FUNCTION_BLOCK FB_AllocateAreaWithRoundbelt EXTENDS FB_ModeBase_V2 IMPLEMENTS I_UnitState
VAR_INPUT
    INPUT       : REFERENCE TO ST_InputTable;
    OUTPUT      : REFERENCE TO ST_OutputTable;
    CurrentData : ST_SetupPara;
    // Componets
    Cylinder 	: REFERENCE TO UNI_CylinderList;
    Service  	: REFERENCE TO ST_AllocateService;
    Motor    	: REFERENCE TO UNI_MotorList;
    Reset       : REFERENCE TO BOOL;
	Stop 		: REFERENCE TO BOOL;
	bStopMem 	: REFERENCE TO BOOL;
END_VAR
VAR_OUTPUT
	Homed : BOOL;
END_VAR
VAR
	Abort	: BOOL;

	// 連動暫停 - 任一 Service 錯誤時暫停所有其他 Service
	_bAnyServiceError : BOOL;

    InitDone          : BOOL;
    Clip              : U_Cylinders;
    Cylinders         : U_Cylinders;
    OutRobotCylinders : Uni_DuoCylinders;
    OutRobotClips     : Uni_DuoCylinders;

    i : INT;
    //============== Service====================
    // Allocate Home
    fbAllocateHome : FB_AllocateAreaHome;
    //RoundBelt
    RoundBeltControl  : FB_RoundBeltService;
    _RoundBeltMoveJob : st_AllocateCircleMoveStructure;
    //RoundBeltMoveJob_Internal 	: st_AllocateCircleMoveStructure;		
    RoundBeltControlAccess               : E_RoundBeltControlAccess := E_RoundBeltControlAccess.Host;
    RoundBeltMoveJob_Ctrl                : ST_CommandBasic;
    RoundBeltMoveJob_Ctrl_Batch          : ST_CommandBasic;
    RoundBeltMoveJob_Status              : ST_StatusBasic;
    RoundBeltMoveJob_Position            : LREAL;
    RoundBeltMoveJob_Position_FanucRobot : LREAL;
    //TurnTable
    TurnTableControl : FB_TurnTableService;

    //Allocating
    fb_AllocateBatchMode        : FB_AllocateMoveAutoBatchMode;
    AutoAllocateJobBatch_Ctrl   : st_AllocateMoveAutoBatchMode_Ctrl;
    AutoAllocateJobBatch_Status : st_AllocateMoveAutoBatchMode_Status;
    bAutoAllocateJobDryRun      : BOOL;

	  //Allocating reverse
    fb_AllocateBatchMode_Reverse        : FB_AllocateMoveAutoBatchMode_Reverse;
    AutoAllocateJobBatch_Reverse_Ctrl   : st_AllocateMoveAutoBatchMode_Ctrl;
    AutoAllocateJobBatch_Reverse_Status : st_AllocateMoveAutoBatchMode_Status;
   
	
    //OutRobot EmptyBoxMove
    fbOutRobot_EmptyBoxMove        : FB_OutRobot_EmptyBoxMove;
    fbOutRobot_EmptyBoxMove_Ctrl   : ST_CommandBasic;
    fbOutRobot_EmptyBoxMove_Status : ST_StatusBasic;

    //OutRobot RareBoxMove
    fbOutRobot_RareBoxMove        : FB_OutRobot_RareBoxMove;
    fbOutRobot_RareBoxMove_Ctrl   : ST_CommandBasic;
    fbOutRobot_RareBoxMove_Status : ST_StatusBasic;

    //OutRobot BoxMoveReverse	
    fbOutRobot_BoxMoveReverse        : FB_OutRobot_BoxMoveReverse;
    fbOutRobot_BoxMoveReverse_Ctrl   : ST_CommandBasic;
    fbOutRobot_BoxMoveReverse_Status : ST_StatusBasic;

	//OutRobot TurnTable to RoundBelt
	fbOutRobot_TurnTableToRoundBelt: FB_OutRobot_BoxMoveTurnTableToRoundBelt;
	fbOutRobot_TurnTableToRoundBel_Ctrl   : ST_CommandBasic;
    fbOutRobot_TurnTableToRoundBel_Status : ST_StatusBasic;
	
    //TransCV Camera
    fbSameSizeCVCamera  		: FB_SameSizeCVCamera;
	fbSameSizeCVCamera_Reverse 	: FB_SameSizeCVCamera_Reverse;
    fbDifferentCVCamera 		: FB_DifferentCVCamera;
	// 逆向拍照批次入料
	fbReverseBatchPickAndPhoto 	: FB_SameSizeCV_ReverseBatchPickAndPhoto;
	fbReverseBoxToWareHouse    	: FB_SameSizeCV_ReverseBoxToWareHouse;
	TransCV_Press 				: BOOL :=FALSE;

    // Round belt
    AutoRotatebelt_Internal_Ctrl   : st_RoundBeltAutoSingleMove_Ctrl;
    AutoRotatebelt_Internal_Status : st_RoundBeltAutoSingleMove_Status;
    _AutoRotatebelt_Ctrl           : st_RoundBeltAutoSingleMove_Ctrl;
    _AutoRotatebelt_Status         : st_RoundBeltAutoSingleMove_Status;
    bInternalRotateBeltRequest     : BOOL;
    bReloadRotateBeltRequest       : BOOL;

    // Pullout

    fbPulloutCV                 : FB_PullOutConveyorAction;
    _AutoPullout_Ctrl           : ST_AutoPullOutConveyorCommand;
    _AutoPullout_Status         : ST_AutoPullOutConveyorSatus;
    _AutoPullout_Info           : ST_PullOutConveyorInfo;
    AutoPullout_Internal_Ctrl   : ST_AutoPullOutConveyorCommand;
    AutoPullout_Internal_Status : ST_AutoPullOutConveyorSatus;
    AutoPullout_Internal_Info   : ST_PullOutConveyorInfo;
    RobotPullout_Internal_Ctrl   : ST_AutoPullOutConveyorCommand;
    RobotPullout_Internal_Status : ST_AutoPullOutConveyorSatus;
    RobotPullout_Internal_Info   : ST_PullOutConveyorInfo;
	fbPulloutCV_BTNCtrl			:FB_PullOutConveyorBtnCtrl;

    PulloutControlAccess        : E_RoundBeltControlAccess := E_RoundBeltControlAccess.Host;
    bPulloutConveyorInternCtrl  : BOOL;
	
	// TurnTable
	 _TurnTableMove                      :  st_ads_OneAxisMoveWithPosition;
	 
	 //AllocateRobotNeedlingMove
	 fbAllocateRobotNeedlingMove		: FB_AllocateRobotNeedlingMove;

END_VAR

SUPER^();
IF __ISVALIDREF(PackTag)  THEN
	
    eModeCommand  := PackTag.Command.UnitMode;
    eStateCommand := PackTag.Command.CntrlCmd;
ELSE
    RETURN;
END_IF

IF __ISVALIDREF(Cylinder) THEN
	
	Clip.stCylinders.Cylinder0 REF= Cylinder.List.fbAllocateRobot_LeftClamp1;
	Clip.stCylinders.Cylinder1 REF= Cylinder.List.fbAllocateRobot_LeftClamp2;
	Clip.stCylinders.Cylinder2 REF= Cylinder.List.fbAllocateRobot_RightClamp1;
	Clip.stCylinders.Cylinder3 REF= Cylinder.List.fbAllocateRobot_RightClamp2;
	Cylinders.stCylinders.Cylinder0 REF= Cylinder.List.fbAllocateRobot_LeftVert1;
	Cylinders.stCylinders.Cylinder1 REF= Cylinder.List.fbAllocateRobot_LeftVert2;
	Cylinders.stCylinders.Cylinder2 REF= Cylinder.List.fbAllocateRobot_RightVert1;
	Cylinders.stCylinders.Cylinder3 REF= Cylinder.List.fbAllocateRobot_RightVert2;
	
	OutRobotCylinders.stCylinders.Cylinder1 REF= Cylinder.List.fbOutRobot_AsideVert;
	OutRobotCylinders.stCylinders.Cylinder2 REF= Cylinder.List.fbOutRobot_BsideVert;
	OutRobotClips.stCylinders.Cylinder1 REF= Cylinder.List.fbOutRobot_AsideClamp;
	OutRobotClips.stCylinders.Cylinder2 REF= Cylinder.List.fbOutRobot_BsideClamp;
	
END_IF

ACTION A00_Service:
// ============================================================================
// 連動暫停邏輯 - 任一 Service 錯誤時，暫停所有其他 Service
// ============================================================================
_bAnyServiceError := FALSE;
//	_RoundBeltMoveJob.HandShake.Error OR
//	_TurnTableMove.HandShake.Error OR
//	AutoAllocateJobBatch_Status.bError OR
//	AutoAllocateJobBatch_Reverse_Status.bError OR
//	Service.AutoMode_EmptyBoxMove.HandShake.Error OR
//	Service.AutoMode_RareBoxMove.HandShake.Error OR
//	Service.AutoMode_BoxMoveReverse.HandShake.Error OR
//	Service.AutoMode_DifferentCVCamera.Status.Error OR
//	fbOutRobot_TurnTableToRoundBel_Status.Error OR
//	Service.AutoMode_SameSizeCVCamera.Status.Error OR
//	_AutoPullout_Status.Error OR
//	Service.AllocateRobotNeedlingMove.Status.Error;

fbAllocateHome(
	xDone=> ,
	xBusy=> ,
	xError=> ,
	xExecute:= ,
	xAbort:= THIS^.Abort OR _bAnyServiceError,
	Homed := Homed,
	Cylinder:= Cylinder, 
	Motor:= Motor, 
	CurrentData:= CurrentData, 
	TimeOut:= , 
	xAborted=> , 
	iErrorID=> , 
	ErrorMsg=> ,
	AxisHomingRequest =>);
	//Service.AllocateRegionHome.Homed:= bHomed;

RoundBeltControl(
	xDone=> _RoundBeltMoveJob.HandShake.Done,
	xBusy=> _RoundBeltMoveJob.HandShake.Busy,
	xError=> _RoundBeltMoveJob.HandShake.Error,
	xExecute:= _RoundBeltMoveJob.HandShake.Execute,
	xAbort:= THIS^.Abort OR _bAnyServiceError,
	TargetStation:= LREAL_TO_INT( _RoundBeltMoveJob.Position),
	Cylinder:= Cylinder, 
	TimeOut:= , 
	xAborted=> , 
	iErrorID=> , 
	ErrorMsg=> ,
	AxisRoundMoveRequest => ,
	Pause	:= bStopMem);
	
TurnTableControl(
	xDone=> _TurnTableMove.HandShake.Done,
	xBusy=> _TurnTableMove.HandShake.Busy,
	xError=> _TurnTableMove.HandShake.Error,
	xExecute:= _TurnTableMove.HandShake.Execute,
	xAbort:= THIS^.Abort OR _bAnyServiceError,
	iTurnTableTarget:= LREAL_TO_INT(_TurnTableMove.Position),
	Cylinder:= Cylinder, 
	//TimeOut:= , 
	xAborted=> , 
	iErrorID=> , 
	ErrorMsg=> ,
	bTurnTableMoveRequest=>,
	Pause := bStopMem);
	
fb_AllocateBatchMode(
	Execute:= AutoAllocateJobBatch_Ctrl.bExecute,
	Abort:= THIS^.Abort OR _bAnyServiceError,
	Reset:= Reset,
	ObjectName:= 'Allocate One process',
	Busy=> AutoAllocateJobBatch_Status.bBusy,
	Done=> AutoAllocateJobBatch_Status.bDone,
	Aborted=> ,
	Error=> AutoAllocateJobBatch_Status.bError,
	ErrorID=>AutoAllocateJobBatch_Status.ErrorID ,
	Status=>AutoAllocateJobBatch_Status.Status ,
	UniqueErrorCode=> , 
	SimpleAllocateMode:= AutoAllocateJobBatch_Ctrl.bSimpleAllocation, 
	bOccupied:=AutoAllocateJobBatch_Ctrl.bOccupied, 
	Clips:= Clip.Cylinders, 
	cylinders:= Cylinders.Cylinders, 
	TurnTable_Press:= Cylinder.List.fbTurntable_Press, 
	RoundBelt_Press:= Cylinder.List.fbRoundBelt_WorkZone_Press, 
	AutoAllocateJobBatch_Ctrl:= AutoAllocateJobBatch_Ctrl, 
	INPUT:= INPUT, 
	OUTPUT:= OUTPUT, 
	NrOfAllocateCylinder:= 4, 
	CurrentData:= CurrentData, 
	bAutoAllocateJobDryRun:= bAutoAllocateJobDryRun, // Dry run : No round belt move
	ProcessedIndex=> AutoAllocateJobBatch_Status.iIndex,
	RoundBeltMoveJob_Ctrl =>,
	RoundBeltMoveJob_Status := RoundBeltMoveJob_Status,
	RoundBeltMoveJob_Position =>	 ,
	Pause := bStopMem);
	
	IF fb_AllocateBatchMode.SimpleAllocateMode THEN
		 Service.AutoMode_SimpleAllocation_Batch.WorkedID:= AutoAllocateJobBatch_Status.iIndex;
	ELSE
		 Service.AutoMode_AllocateBatchMode.WorkedID:= AutoAllocateJobBatch_Status.iIndex;
	END_IF
fb_AllocateBatchMode_Reverse(
	Execute:=AutoAllocateJobBatch_Reverse_Ctrl.bExecute ,
	Abort:= THIS^.Abort OR _bAnyServiceError,
	Reset:= Reset,
	Pause:= bStopMem,
	ObjectName:= 'Allocate batch reverse',
	Busy=> AutoAllocateJobBatch_Reverse_Status.bBusy,
	Done=> AutoAllocateJobBatch_Reverse_Status.bDone,
	Aborted=> AutoAllocateJobBatch_Reverse_Status.bAborted,
	Error=> AutoAllocateJobBatch_Reverse_Status.bError,
	ErrorID=> AutoAllocateJobBatch_Reverse_Status.ErrorID,
	Status=> AutoAllocateJobBatch_Reverse_Status.Status,
	UniqueErrorCode=> ,  
	bOccupied:= AutoAllocateJobBatch_Reverse_Ctrl.bOccupied, 
	Clips:= Clip.Cylinders, 
	cylinders:= Cylinders.Cylinders, 
	TurnTable_Press:= Cylinder.List.fbTurntable_Press, 
	RoundBelt_Press:= Cylinder.List.fbRoundBelt_WorkZone_Press, 
	AutoAllocateJobBatch_Reverse_Ctrl:= AutoAllocateJobBatch_Reverse_Ctrl, 
	INPUT:= INPUT, 
	OUTPUT:= OUTPUT, 
	NrOfAllocateCylinder:=4 , 
	CurrentData:= CurrentData, 
	bAutoAllocateJobDryRun:= bAutoAllocateJobDryRun, 
	RoundBeltMoveJob_Ctrl=> , 
	ProcessedIndex=> AutoAllocateJobBatch_Reverse_Status.iIndex,
	RoundBeltMoveJob_Status := RoundBeltMoveJob_Status,
	RoundBeltMoveJob_Position =>);

	
fbOutRobot_EmptyBoxMove(
	Execute:= Service.AutoMode_EmptyBoxMove.HandShake.Execute,
	Abort:= THIS^.Abort OR _bAnyServiceError,
	Reset:= Reset ,
	ObjectName:= 'fbOutRobot_EmptyBoxMove', 
	Busy=> Service.AutoMode_EmptyBoxMove.HandShake.Busy, 
	Done=> Service.AutoMode_EmptyBoxMove.HandShake.Done, 
	Aborted=> , 
	Error=> Service.AutoMode_EmptyBoxMove.HandShake.Error, 
	ErrorID=> , 
	Status=> , 
	UniqueErrorCode=> , 
	INPUT:= INPUT, 
	Cylinder:= Cylinder, 
	Motor:= Motor, 
	Cylinders :=OutRobotCylinders.Cylinders,
	Clips := OutRobotClips.Cylinders,
	AutoMode_OutRobotMoveMove:=Service.AutoMode_EmptyBoxMove );

fbOutRobot_RareBoxMove(
	Execute:= Service.AutoMode_RareBoxMove.HandShake.Execute ,
	Abort:= THIS^.Abort OR _bAnyServiceError,
	Reset:= Reset,
	ObjectName:= 'fbOutRobot_RareBoxMove', 
	Busy=> Service.AutoMode_RareBoxMove.HandShake.Busy, 
	Done=> Service.AutoMode_RareBoxMove.HandShake.Done, 
	Aborted=> , 
	Error=> Service.AutoMode_RareBoxMove.HandShake.Error, 
	ErrorID=> , 
	Status=> , 
	UniqueErrorCode=> , 
	INPUT:=INPUT , 
	Cylinder:= Cylinder, 
	Motor:= Motor, 
	Cylinders :=OutRobotCylinders.Cylinders,
	Clips := OutRobotClips.Cylinders,
	AutoMode_OutRobotMoveMove:= Service.AutoMode_RareBoxMove);

fbOutRobot_BoxMoveReverse(
	Execute:= Service.AutoMode_BoxMoveReverse.HandShake.Execute,
	Abort:= THIS^.Abort OR _bAnyServiceError,
	Reset:= Reset,
	ObjectName:='fbOutRobot_BoxMoveReverse', 
	Busy=> Service.AutoMode_BoxMoveReverse.HandShake.Busy, 
	Done=> Service.AutoMode_BoxMoveReverse.HandShake.Done, 
	Aborted=> , 
	Error=> Service.AutoMode_BoxMoveReverse.HandShake.Error, 
	ErrorID=> , 
	Status=> , 
	UniqueErrorCode=> , 
	INPUT:= INPUT, 
	Cylinder:= Cylinder, 
	Motor:= Motor, 
	Cylinders :=OutRobotCylinders.Cylinders,
	Clips := OutRobotClips.Cylinders,
	AutoMode_OutRobotMoveMove:= Service.AutoMode_BoxMoveReverse,
	pause := bStopMem);	
	
fbDifferentCVCamera(
	xDone=> Service.AutoMode_DifferentCVCamera.Status.Done,
	xBusy=> Service.AutoMode_DifferentCVCamera.Status.Busy,
	xError=> Service.AutoMode_DifferentCVCamera.Status.Error,
	xExecute:= Service.AutoMode_DifferentCVCamera.Command.Execute,
	xAbort:= Service.AutoMode_DifferentCVCamera.Command.Abort OR THIS^.Abort OR _bAnyServiceError,
	xReset:= Reset,
	Cylinder:= Cylinder, 
	TimeOut:= , 
	Input:= INPUT, 
	OutPut:= OutPut ,
	Motor:= Motor, 
	BoxCameraDone:= Service.AutoMode_DifferentCVCamera.BoxCameraDone, 
	xAborted=> , 
	iErrorID=> , 
	ErrorMsg=> , 
	UseBoxCamera=> Service.AutoMode_DifferentCVCamera.UseBoxCamera);

fbOutRobot_TurnTableToRoundBelt(
	Execute:= fbOutRobot_TurnTableToRoundBel_Ctrl.Execute,
	Abort:= fbOutRobot_TurnTableToRoundBel_Ctrl.Abort OR THIS^.Abort OR _bAnyServiceError,
	Reset:= Reset,
	ObjectName:= 'fbOutRobot_TurnTableToRoundBelt', 
	Busy=> fbOutRobot_TurnTableToRoundBel_Status.Busy, 
	Done=> fbOutRobot_TurnTableToRoundBel_Status.Done, 
	Aborted=> , 
	Error=> fbOutRobot_TurnTableToRoundBel_Status.Error, 
	ErrorID=> , 
	Status=> fbOutRobot_TurnTableToRoundBel_Status.Status, 
	UniqueErrorCode=> , 
	INPUT:= INPUT, 
	Cylinders:= OutRobotCylinders.Cylinders, 
	Clips:=OutRobotClips.Cylinders , 
	AutoMode_TurnTableToRoundBelt:= ); // todo creative var to fill in cmooand info	
	
	fbSameSizeCVCamera(
		xReset := Reset,
		xDone=> Service.AutoMode_SameSizeCVCamera.Status.Done,
		xBusy=> Service.AutoMode_SameSizeCVCamera.Status.Busy,
		xError=> Service.AutoMode_SameSizeCVCamera.Status.Error,
		xExecute:= Service.AutoMode_SameSizeCVCamera.Command.Execute,
		xAbort:= Service.AutoMode_SameSizeCVCamera.Command.Abort OR THIS^.Abort OR _bAnyServiceError,
		Cylinder:= Cylinder, 
		TimeOut:= , 
		Input:= INPUT, 
		OutPut:= OUTPUT, 
		Motor:= Motor, 
		BoxCameraDone:= Service.AutoMode_SameSizeCVCamera.BoxCameraDone, 
		xAborted=> , 
		iErrorID=> , 
		ErrorMsg=> , 
		UseBoxCamera=> Service.AutoMode_SameSizeCVCamera.UseBoxCamera);
		
	fbSameSizeCVCamera_Reverse(
		xReset := Service.AutoMode_SameSizeCVCamera_Reverse.Command.Reset,
		xDone=> Service.AutoMode_SameSizeCVCamera_Reverse.Status.Done,
		xBusy=> Service.AutoMode_SameSizeCVCamera_Reverse.Status.Busy,
		xError=> Service.AutoMode_SameSizeCVCamera_Reverse.Status.Error,
		xExecute:= Service.AutoMode_SameSizeCVCamera_Reverse.Command.Execute,
		xAbort:= Service.AutoMode_SameSizeCVCamera_Reverse.Command.Abort OR THIS^.Abort OR _bAnyServiceError,
		Cylinder:= Cylinder,
		TimeOut:= ,
		Input:= INPUT,
		OutPut:= OUTPUT,
		Motor:= Motor,
		BoxCameraDone:= Service.AutoMode_SameSizeCVCamera_Reverse.BoxCameraDone,
		xAborted=> ,
		iErrorID=> ,
		ErrorMsg=> ,
		UseBoxCamera=> Service.AutoMode_SameSizeCVCamera_Reverse.UseBoxCamera);
		
	// ================================================================
	// 逆向拍照批次入料 — 逐欄位 link ADS HandShake
	// ================================================================

	// --- fbReverseBoxToWareHouse (子FB: 軌道→大手臂→入倉/NG，輸送帶要先動) ---
	fbReverseBoxToWareHouse(
		// Command (C# → PLC)
		Execute := Service.AutoMode_ReverseBoxToWareHouse.Command.Execute,
		Abort := Service.AutoMode_ReverseBoxToWareHouse.Command.Abort OR THIS^.Abort OR _bAnyServiceError,
		Reset := Service.AutoMode_ReverseBoxToWareHouse.Command.Reset,
		ObjectName := 'Reverse box to warehouse',
		// 盒子資訊 (C# → PLC)
		bBoxA_Enable := Service.AutoMode_ReverseBoxToWareHouse.bBoxA_Enable,
		bBoxA_IsOK := Service.AutoMode_ReverseBoxToWareHouse.bBoxA_IsOK,
		iBoxA_Warehouse := Service.AutoMode_ReverseBoxToWareHouse.iBoxA_Warehouse,
		iBoxA_Level := Service.AutoMode_ReverseBoxToWareHouse.iBoxA_Level,
		iBoxA_Track := Service.AutoMode_ReverseBoxToWareHouse.iBoxA_Track,
		bBoxB_Enable := Service.AutoMode_ReverseBoxToWareHouse.bBoxB_Enable,
		bBoxB_IsOK := Service.AutoMode_ReverseBoxToWareHouse.bBoxB_IsOK,
		iBoxB_Warehouse := Service.AutoMode_ReverseBoxToWareHouse.iBoxB_Warehouse,
		iBoxB_Level := Service.AutoMode_ReverseBoxToWareHouse.iBoxB_Level,
		iBoxB_Track := Service.AutoMode_ReverseBoxToWareHouse.iBoxB_Track,
		// 硬體
		Cylinder := Cylinder,
		Motor := Motor,
		Input := INPUT,
		OutPut := OUTPUT,
		StorageRobot := DAS_CoreSys.MachineControl.FanucRobot.List.StorageRobot,
		WareHouse := DAS_CoreSys.MachineControl.fbStorageArea.fbWarehouse,
		Stop := bStopMem,
		// Status output (PLC → C#)
		bBoxA_Done => Service.AutoMode_ReverseBoxToWareHouse.bBoxA_Done,
		bBoxB_Done => Service.AutoMode_ReverseBoxToWareHouse.bBoxB_Done);
	// Status (PLC → C#)
	Service.AutoMode_ReverseBoxToWareHouse.Status.Done	:= fbReverseBoxToWareHouse.Done;
	Service.AutoMode_ReverseBoxToWareHouse.Status.Busy	:= fbReverseBoxToWareHouse.Busy;
	Service.AutoMode_ReverseBoxToWareHouse.Status.Error	:= fbReverseBoxToWareHouse.Error;	

	// --- fbReverseBatchPickAndPhoto (主FB: 三軌 Pipeline) ---
	fbReverseBatchPickAndPhoto(
		// Command (C# → PLC)
		Execute := Service.AutoMode_ReverseBatchPick.Command.Execute,
		Abort := Service.AutoMode_ReverseBatchPick.Command.Abort OR THIS^.Abort OR _bAnyServiceError,
		Reset := Service.AutoMode_ReverseBatchPick.Command.Reset,
		ObjectName := 'Reverse batch pick and photo',
		// 鐵盤 Sensor (C# → PLC, 後續改硬體訊號)
		bLeftPlateReady := Service.AutoMode_ReverseBatchPick.bLeftPlateReady,
		bRightPlateReady := Service.AutoMode_ReverseBatchPick.bRightPlateReady,
		// 鐵盤配置 (C# → PLC)
		LeftPlate := Service.AutoMode_ReverseBatchPick.LeftPlate,
		RightPlate := Service.AutoMode_ReverseBatchPick.RightPlate,
		bLeftConfigReady := Service.AutoMode_ReverseBatchPick.bLeftConfigReady,
		bRightConfigReady := Service.AutoMode_ReverseBatchPick.bRightConfigReady,
		// 拍照結果 (C# → PLC)
		BoxCameraDone := Service.AutoMode_ReverseBatchPick.BoxCameraDone,
		CameraIsOK := Service.AutoMode_ReverseBatchPick.CameraIsOK,
		CameraWarehouse := Service.AutoMode_ReverseBatchPick.CameraWarehouse,
		CameraLevel := Service.AutoMode_ReverseBatchPick.CameraLevel,
		CameraTrack := Service.AutoMode_ReverseBatchPick.CameraTrack,
		// 硬體
		Cylinder := Cylinder,
		Motor := Motor,
		Input := INPUT,
		OutPut := OUTPUT,
		StorageRobot := DAS_CoreSys.MachineControl.FanucRobot.List.StorageRobot,
		ShippingRobot := DAS_CoreSys.MachineControl.FanucRobot.List.ShippingRobot,
		WareHouse := DAS_CoreSys.MachineControl.fbStorageArea.fbWarehouse,
		Stop := bStopMem,
		// Status output (PLC → C#)
		bLeftPlateArrived => Service.AutoMode_ReverseBatchPick.bLeftPlateArrived,
		bRightPlateArrived => Service.AutoMode_ReverseBatchPick.bRightPlateArrived,
		bLeftPlateDone => Service.AutoMode_ReverseBatchPick.bLeftPlateDone,
		bRightPlateDone => Service.AutoMode_ReverseBatchPick.bRightPlateDone,
		UseBoxCamera => Service.AutoMode_ReverseBatchPick.UseBoxCamera,
		uiUnphotographedCount => Service.AutoMode_ReverseBatchPick.uiUnphotographedCount,
		uiTotalProcessed => Service.AutoMode_ReverseBatchPick.uiTotalProcessed,
		uiTransportedCount => Service.AutoMode_ReverseBatchPick.uiTransportedCount);
	// Status (PLC → C#)
	Service.AutoMode_ReverseBatchPick.Status.Done	:= fbReverseBatchPickAndPhoto.Done;
	Service.AutoMode_ReverseBatchPick.Status.Busy	:= fbReverseBatchPickAndPhoto.Busy;
	Service.AutoMode_ReverseBatchPick.Status.Error	:= fbReverseBatchPickAndPhoto.Error;

	
fbPulloutCV(
	Execute:= _AutoPullout_Ctrl.Execute,
	Abort:= _AutoPullout_Ctrl.Abort OR THIS^.Abort OR _bAnyServiceError,
	Reset:= Reset,
	ObjectName:= ' Pullout conveyor ', 
	Busy=> _AutoPullout_Status.Busy, 
	Done=> _AutoPullout_Status.Done, 
	Aborted=> , 
	Error=> _AutoPullout_Status.Error, 
	ErrorID=> , 
	Status=> _AutoPullout_Status.Status, 
	UniqueErrorCode=> , 
	FixCylinderA1:= Cylinder.List.fbPullOutCV_AsidePress1, 
	FixCylinderA2:= Cylinder.List.fbPullOutCV_AsidePress2, 
	FixCylinderB1:= Cylinder.List.fbPullOutCV_BsidePress1, 
	FixCylinderB2:= Cylinder.List.fbPullOutCV_BsidePress2, 
	BarrierCylinderA:= Cylinder.List.fbPullOutCV_AsideBlock, 
	BarrierCylinderB:= Cylinder.List.fbPullOutCV_BsideBlock, 
	ConveyorMotorA:= Motor.List.PullOutCV_A, 
	ConveyorMotorB:= Motor.List.PullOutCV_B, 
	INPUT:= INPUT, 
	PullOutInfo:= _AutoPullout_Info);
	
fbPulloutCV_BTNCtrl(
	Input:= INPUT, 
	Output:= OUTPUT, 
	Motor:= Motor, 
	bPullOutConveyorExecute:= _AutoPullout_Ctrl.Execute, 
	bPullOutConveyorDone:= _AutoPullout_Status.Done, 
	bPullOutConveyorBusy:= _AutoPullout_Status.Busy, 
	StroageRegionMode:= eModeCurrent, 
	PullOutConveyorState=> );
	
fbAllocateRobotNeedlingMove(
	xDone=>  Service.AllocateRobotNeedlingMove.Status.Done,
	xBusy=> Service.AllocateRobotNeedlingMove.Status.Busy,
	xError=> Service.AllocateRobotNeedlingMove.Status.Error,
	xExecute:= Service.AllocateRobotNeedlingMove.Command.Execute,
	xAbort:= Service.AllocateRobotNeedlingMove.Command.Abort OR THIS^.Abort OR _bAnyServiceError,
	TimeOut:= , 
	MovingInfo:= Service.AllocateRobotNeedlingMove.MovingInfo, 
	xAborted=> , 
	iErrorID=> , 
	ErrorMsg=> Service.AllocateRobotNeedlingMove.Status.Status);
END_ACTION

ACTION A01_RoundBeltAccessControl:
CASE RoundBeltControlAccess OF 
	E_RoundBeltControlAccess.Host :
	 IF eModeCurrent = E_UnitMode.Manual THEN
		_RoundBeltMoveJob.Position :=Service.AllocateCircleMove.Position;
		_RoundBeltMoveJob.Latch :=Service.AllocateCircleMove.Latch;
		_RoundBeltMoveJob.HandShake.Execute :=Service.AllocateCircleMove.HandShake.Execute;
		_RoundBeltMoveJob.HandShake.Reset :=Service.AllocateCircleMove.HandShake.Reset;
		_RoundBeltMoveJob.HandShake.Occupied  :=Service.AllocateCircleMove.HandShake.Occupied;
		Service.AllocateCircleMove.HandShake.Busy := _RoundBeltMoveJob.HandShake.Busy;
		Service.AllocateCircleMove.HandShake.Done := _RoundBeltMoveJob.HandShake.Done;
		Service.AllocateCircleMove.HandShake.Error := _RoundBeltMoveJob.HandShake.Error;
	ELSIF  eModeCurrent = E_UnitMode.Auto THEN
		_RoundBeltMoveJob.Position :=Service.AutoMode_AllocateCircleMove.Position;
		_RoundBeltMoveJob.Latch :=Service.AutoMode_AllocateCircleMove.Latch;
		_RoundBeltMoveJob.HandShake.Execute :=Service.AutoMode_AllocateCircleMove.HandShake.Execute;
		_RoundBeltMoveJob.HandShake.Reset :=Service.AutoMode_AllocateCircleMove.HandShake.Reset;
		_RoundBeltMoveJob.HandShake.Occupied  :=Service.AutoMode_AllocateCircleMove.HandShake.Occupied;
		Service.AutoMode_AllocateCircleMove.HandShake.Busy := _RoundBeltMoveJob.HandShake.Busy;
		Service.AutoMode_AllocateCircleMove.HandShake.Done := _RoundBeltMoveJob.HandShake.Done;
		Service.AutoMode_AllocateCircleMove.HandShake.Error := _RoundBeltMoveJob.HandShake.Error;
	END_IF
		
	E_RoundBeltControlAccess.Allocating  :
	
		_RoundBeltMoveJob.Position :=RoundBeltMoveJob_Position;
		//_RoundBeltMoveJob.Latch :=;
		_RoundBeltMoveJob.HandShake.Execute :=RoundBeltMoveJob_Ctrl_Batch.Execute;
		_RoundBeltMoveJob.HandShake.Reset :=RoundBeltMoveJob_Ctrl_Batch.Reset;
		RoundBeltMoveJob_Status.Busy := _RoundBeltMoveJob.HandShake.Busy;
		RoundBeltMoveJob_Status.Done := _RoundBeltMoveJob.HandShake.Done;
		RoundBeltMoveJob_Status.Error := _RoundBeltMoveJob.HandShake.Error;

	E_RoundBeltControlAccess.FanucRobot:
		_RoundBeltMoveJob.Position :=RoundBeltMoveJob_Position_FanucRobot;
		//_RoundBeltMoveJob.Latch :=;
		_RoundBeltMoveJob.HandShake.Execute :=RoundBeltMoveJob_Ctrl.Execute;
		_RoundBeltMoveJob.HandShake.Reset :=RoundBeltMoveJob_Ctrl.Reset;
		RoundBeltMoveJob_Status.Busy := _RoundBeltMoveJob.HandShake.Busy;
		RoundBeltMoveJob_Status.Done := _RoundBeltMoveJob.HandShake.Done;
		RoundBeltMoveJob_Status.Error := _RoundBeltMoveJob.HandShake.Error;	
END_CASE
END_ACTION

ACTION A02_PulloutAccessControl:
CASE PulloutControlAccess OF
    E_RoundBeltControlAccess.Host:
        _AutoPullout_Ctrl.Execute := Service.AutoMode_PullOutConveyor.Command.Execute;
        _AutoPullout_Ctrl.Abort := Service.AutoMode_PullOutConveyor.Command.Abort;
        _AutoPullout_Ctrl.Reset := Service.AutoMode_PullOutConveyor.Command.Reset;
        Service.AutoMode_PullOutConveyor.Status.Busy := _AutoPullout_Status.Busy;
        Service.AutoMode_PullOutConveyor.Status.Done := _AutoPullout_Status.Done;
        Service.AutoMode_PullOutConveyor.Status.Error := _AutoPullout_Status.Error;
        Service.AutoMode_PullOutConveyor.Status.Status := _AutoPullout_Status.Status;
        _AutoPullout_Info := Service.AutoMode_PullOutConveyor.PullOutConveyorInfo;
    E_RoundBeltControlAccess.Allocating:
        _AutoPullout_Ctrl.Execute := AutoPullout_Internal_Ctrl.Execute;
        _AutoPullout_Ctrl.Abort := AutoPullout_Internal_Ctrl.Abort;
        _AutoPullout_Ctrl.Reset := AutoPullout_Internal_Ctrl.Reset;
        AutoPullout_Internal_Status.Busy := _AutoPullout_Status.Busy;
        AutoPullout_Internal_Status.Done := _AutoPullout_Status.Done;
        AutoPullout_Internal_Status.Error := _AutoPullout_Status.Error;
        AutoPullout_Internal_Status.Status := _AutoPullout_Status.Status;
        _AutoPullout_Info := AutoPullout_Internal_Info;
    E_RoundBeltControlAccess.FanucRobot:
        _AutoPullout_Ctrl.Execute := RobotPullout_Internal_Ctrl.Execute;
        _AutoPullout_Ctrl.Abort := RobotPullout_Internal_Ctrl.Abort;
        _AutoPullout_Ctrl.Reset := RobotPullout_Internal_Ctrl.Reset;
        RobotPullout_Internal_Status.Busy := _AutoPullout_Status.Busy;
        RobotPullout_Internal_Status.Done := _AutoPullout_Status.Done;
        RobotPullout_Internal_Status.Error := _AutoPullout_Status.Error;
        RobotPullout_Internal_Status.Status := _AutoPullout_Status.Status;
        _AutoPullout_Info := RobotPullout_Internal_Info;
END_CASE
END_ACTION

ACTION A99_ErrorHandler:

END_ACTION

METHOD M_Aborted
Abort := FALSE;
M_StateComplete();
END_METHOD

METHOD M_Aborting
Abort := TRUE;
M_StateComplete();
END_METHOD

METHOD M_ActiveRoundBeltInternalCtrl : BOOL
VAR_INPUT
END_VAR
bReloadRotateBeltRequest := TRUE;
M_ActiveRoundBeltInternalCtrl := true; // Method end
END_METHOD

METHOD PRIVATE M_AutoAllocatingBatch : BOOL
VAR_INPUT
END_VAR
IF NOT Service.AutoMode_SimpleAllocation_Batch.HandShake.Execute 
   AND NOT Service.AutoMode_SimpleAllocation_Batch.HandShake.Busy
   AND NOT Service.AutoMode_AllocateBatchMode_Reverse.HandShake.Execute
   AND NOT Service.AutoMode_AllocateBatchMode_Reverse.HandShake.Busy THEN
	
	AutoAllocateJobBatch_Ctrl.bSimpleAllocation:=FALSE;
	AutoAllocateJobBatch_Ctrl.bExecute:=Service.AutoMode_AllocateBatchMode.HandShake.Execute;
	AutoAllocateJobBatch_Ctrl.bReset :=Service.AutoMode_AllocateBatchMode.HandShake.Reset;
	AutoAllocateJobBatch_Ctrl.bOccupied:=Service.AutoMode_AllocateBatchMode.HandShake.Occupied;
	AutoAllocateJobBatch_Ctrl.bPause :=Service.AutoMode_AllocateBatchMode.Pause;

	AutoAllocateJobBatch_Ctrl.AutoMode_AllocateMoveBatch.AllocationInfo:=Service.AutoMode_AllocateBatchMode.AllocationInfo;
	AutoAllocateJobBatch_Ctrl.AutoMode_AllocateMoveBatch.NrOfAllocationJob:=Service.AutoMode_AllocateBatchMode.NrOfAllocationJob;

	Service.AutoMode_AllocateBatchMode.WorkedID:=AutoAllocateJobBatch_Ctrl.AutoMode_AllocateMoveBatch.WorkedID;
	Service.AutoMode_AllocateBatchMode.HandShake.Busy:= AutoAllocateJobBatch_Status.bBusy;
	Service.AutoMode_AllocateBatchMode.HandShake.Error:= AutoAllocateJobBatch_Status.bError;
	Service.AutoMode_AllocateBatchMode.HandShake.Done:= AutoAllocateJobBatch_Status.bDone;
	
	RoundBeltMoveJob_Ctrl_Batch :=fb_AllocateBatchMode.RoundBeltMoveJob_Ctrl; 
	RoundBeltMoveJob_Position :=fb_AllocateBatchMode.RoundBeltMoveJob_Position;	
	bAutoAllocateJobDryRun := FALSE;
END_IF
END_METHOD

METHOD PRIVATE M_AutoAllocatingBatch_Reverse : BOOL
VAR_INPUT
END_VAR
IF NOT Service.AutoMode_AllocateBatchMode.HandShake.Execute 
   AND NOT Service.AutoMode_AllocateBatchMode.HandShake.Busy
   AND NOT Service.AutoMode_SimpleAllocation_Batch.HandShake.Execute
   AND NOT Service.AutoMode_SimpleAllocation_Batch.HandShake.Busy THEN
	AutoAllocateJobBatch_Reverse_Ctrl.bExecute:=Service.AutoMode_AllocateBatchMode_Reverse.HandShake.Execute;
	AutoAllocateJobBatch_Reverse_Ctrl.bReset :=Service.AutoMode_AllocateBatchMode_Reverse.HandShake.Reset;
	AutoAllocateJobBatch_Reverse_Ctrl.bOccupied:=Service.AutoMode_AllocateBatchMode_Reverse.HandShake.Occupied;
	AutoAllocateJobBatch_Reverse_Ctrl.bPause :=Service.AutoMode_AllocateBatchMode_Reverse.Pause;

	AutoAllocateJobBatch_Reverse_Ctrl.AutoMode_AllocateMoveBatch.AllocationInfo:=Service.AutoMode_AllocateBatchMode_Reverse.AllocationInfo;
	AutoAllocateJobBatch_Reverse_Ctrl.AutoMode_AllocateMoveBatch.NrOfAllocationJob:=Service.AutoMode_AllocateBatchMode_Reverse.NrOfAllocationJob;

	Service.AutoMode_AllocateBatchMode_Reverse.WorkedID:=AutoAllocateJobBatch_Reverse_Ctrl.AutoMode_AllocateMoveBatch.WorkedID;
	Service.AutoMode_AllocateBatchMode_Reverse.HandShake.Busy:= AutoAllocateJobBatch_Reverse_Status.bBusy;
	Service.AutoMode_AllocateBatchMode_Reverse.HandShake.Error:= AutoAllocateJobBatch_Reverse_Status.bError;
	Service.AutoMode_AllocateBatchMode_Reverse.HandShake.Done:= AutoAllocateJobBatch_Reverse_Status.bDone;
	RoundBeltMoveJob_Ctrl_Batch :=fb_AllocateBatchMode_Reverse.RoundBeltMoveJob_Ctrl; 
	RoundBeltMoveJob_Position :=fb_AllocateBatchMode_Reverse.RoundBeltMoveJob_Position;	

	bAutoAllocateJobDryRun := FALSE;
	
	END_IF
END_METHOD

METHOD PRIVATE M_AutoAllocatingBatch_Simple : BOOL
VAR_INPUT
END_VAR
IF NOT Service.AutoMode_AllocateBatchMode.HandShake.Execute 
   AND NOT Service.AutoMode_AllocateBatchMode.HandShake.Busy
   AND NOT Service.AutoMode_AllocateBatchMode_Reverse.HandShake.Execute
   AND NOT Service.AutoMode_AllocateBatchMode_Reverse.HandShake.Busy THEN
	
	AutoAllocateJobBatch_Ctrl.bSimpleAllocation:=TRUE;
	AutoAllocateJobBatch_Ctrl.bExecute:=Service.AutoMode_SimpleAllocation_Batch.HandShake.Execute;
	AutoAllocateJobBatch_Ctrl.bReset :=Service.AutoMode_SimpleAllocation_Batch.HandShake.Reset;
	AutoAllocateJobBatch_Ctrl.bOccupied:=Service.AutoMode_SimpleAllocation_Batch.HandShake.Occupied;
	AutoAllocateJobBatch_Ctrl.bPause :=Service.AutoMode_SimpleAllocation_Batch.Pause;

	AutoAllocateJobBatch_Ctrl.AutoMode_AllocateMoveBatch.AllocationInfo:=Service.AutoMode_SimpleAllocation_Batch.AllocationInfo;
	AutoAllocateJobBatch_Ctrl.AutoMode_AllocateMoveBatch.NrOfAllocationJob:=Service.AutoMode_SimpleAllocation_Batch.NrOfAllocationJob;

	Service.AutoMode_SimpleAllocation_Batch.WorkedID:=AutoAllocateJobBatch_Ctrl.AutoMode_AllocateMoveBatch.WorkedID;
	Service.AutoMode_SimpleAllocation_Batch.HandShake.Busy:= AutoAllocateJobBatch_Status.bBusy;
	Service.AutoMode_SimpleAllocation_Batch.HandShake.Error:= AutoAllocateJobBatch_Status.bError;
	Service.AutoMode_SimpleAllocation_Batch.HandShake.Done:= AutoAllocateJobBatch_Status.bDone;
	
	RoundBeltMoveJob_Ctrl_Batch :=fb_AllocateBatchMode.RoundBeltMoveJob_Ctrl; 
	RoundBeltMoveJob_Position :=fb_AllocateBatchMode.RoundBeltMoveJob_Position;		

	bAutoAllocateJobDryRun := FALSE;
END_IF
END_METHOD

METHOD PRIVATE M_AutoTurnTable : BOOL
VAR_INPUT
END_VAR
_TurnTableMove.HandShake.Execute:=Service.AutoMode_TurnTableMove.HandShake.Execute;
_TurnTableMove.Position:=Service.AutoMode_TurnTableMove.Position;

Service.AutoMode_TurnTableMove.HandShake.Busy := _TurnTableMove.HandShake.Busy;
Service.AutoMode_TurnTableMove.HandShake.Done := _TurnTableMove.HandShake.Done;
Service.AutoMode_TurnTableMove.HandShake.Error := _TurnTableMove.HandShake.Error;
END_METHOD

METHOD PRIVATE M_CheckAxesHomed : BOOL
VAR_INPUT
END_VAR

VAR 
	AxisIndex : INT;//1-6
	bCheckHome : BOOL:=TRUE;
END_VAR
bCheckHome:=TRUE;

FOR AxisIndex :=1 TO 6 DO
	bCheckHome:=bCheckHome AND	arAxisCtrl_gb[AxisIndex].Admin.Axis.Status.Homed;
END_FOR

M_CheckAxesHomed:=	bCheckHome;
END_METHOD

METHOD M_Clearing
M_StateComplete();
END_METHOD

METHOD M_Complete
M_StateComplete();
END_METHOD

METHOD M_Completing
M_StateComplete();
END_METHOD

METHOD M_Execute
CASE eModeCurrent OF
	E_UnitMode.Manual:
		M_ManualAllocating();
		M_AutoAllocatingBatch_Simple();
		M_AutoAllocatingBatch();
		M_AutoAllocatingBatch_Reverse();
		M_ManualTurnTable();
		M_AutoAllocatingBatch_Reverse();
		//M_TransCVCameraPress_ManualMode();
		//TransCV_Press :=FALSE;

	E_UnitMode.Auto:
	
		M_AutoAllocatingBatch_Simple();
		M_AutoAllocatingBatch();
		M_AutoAllocatingBatch_Reverse();
		M_AutoTurnTable();
		M_TransCVCameraPress();
END_CASE
//M_StateComplete();
A00_Service();
A01_RoundBeltAccessControl();
A02_PulloutAccessControl();
//bHomed :=M_CheckAxesHomed();
END_METHOD

METHOD PUBLIC M_GetPulloutAccess : BOOL
VAR_INPUT
	 ControlAccess:	 E_RoundBeltControlAccess;
END_VAR
IF THIS^.PulloutControlAccess = E_RoundBeltControlAccess.Host AND 
	NOT (fbPulloutCV.Execute OR fbPulloutCV.Busy OR fbPulloutCV.Done) THEN
	THIS^.PulloutControlAccess := ControlAccess;
	M_GetPulloutAccess := TRUE;
 ELSE
	M_GetPulloutAccess := FALSE;	
 END_IF
END_METHOD

METHOD PUBLIC M_GetRoundBeltAccess : BOOL
VAR_INPUT
	 ControlAccess:	 E_RoundBeltControlAccess;
END_VAR
IF THIS^.RoundBeltControlAccess = E_RoundBeltControlAccess.Host AND 
	NOT (RoundBeltControl.xExecute OR RoundBeltControl.xBusy OR RoundBeltControl.xDone) THEN
	THIS^.RoundBeltControlAccess := ControlAccess;
	M_GetRoundBeltAccess := TRUE;
 ELSE
	M_GetRoundBeltAccess := FALSE;	
 END_IF
END_METHOD

METHOD M_Held
M_StateComplete();
END_METHOD

METHOD M_Holding
M_StateComplete();
END_METHOD

METHOD M_Idle
M_StateComplete();
END_METHOD

METHOD M_InactiveRoundBeltInternalCtrl : BOOL
VAR_INPUT
END_VAR
bReloadRotateBeltRequest := FALSE;

M_InactiveRoundBeltInternalCtrl := true; // Method end
END_METHOD

METHOD PRIVATE M_ManualAllocating : BOOL
VAR_INPUT
END_VAR

VAR_INST 
	
END_VAR

	AutoAllocateJobBatch_Ctrl.bSimpleAllocation:=FALSE;
	AutoAllocateJobBatch_Ctrl.bReset:=Service.AllocateMoveStructure.HandShake.Reset;
	AutoAllocateJobBatch_Ctrl.bPause:=FALSE;
	AutoAllocateJobBatch_Ctrl.bOccupied :=Service.AllocateMoveStructure.HandShake.Occupied;
	AutoAllocateJobBatch_Ctrl.bExecute:=Service.AllocateMoveStructure.HandShake.Execute;
	AutoAllocateJobBatch_Ctrl.AutoMode_AllocateMoveBatch.NrOfAllocationJob:=1;
	AutoAllocateJobBatch_Ctrl.AutoMode_AllocateMoveBatch.AllocationInfo[0].FastMode:=FALSE;
	AutoAllocateJobBatch_Ctrl.AutoMode_AllocateMoveBatch.AllocationInfo[0].SyncMode:=FALSE	;
	
	AutoAllocateJobBatch_Ctrl.AutoMode_AllocateMoveBatch.AllocationInfo[0].PickingNeedleInfo[0].CycleStart:=TRUE;
	AutoAllocateJobBatch_Ctrl.AutoMode_AllocateMoveBatch.AllocationInfo[0].PickingNeedleInfo[0].Box:=LREAL_TO_UINT( Service.AllocateMoveStructure.Frombox);
	AutoAllocateJobBatch_Ctrl.AutoMode_AllocateMoveBatch.AllocationInfo[0].PickingNeedleInfo[0].Clip:=LREAL_TO_INT(Service.AllocateMoveStructure.Clip);
	AutoAllocateJobBatch_Ctrl.AutoMode_AllocateMoveBatch.AllocationInfo[0].PickingNeedleInfo[0].NeedleLocation:=LREAL_TO_INT(Service.AllocateMoveStructure.FromPosition);
	AutoAllocateJobBatch_Ctrl.AutoMode_AllocateMoveBatch.AllocationInfo[0].PlacingNeedleInfo[0].CycleStart:=TRUE;
	
	AutoAllocateJobBatch_Ctrl.AutoMode_AllocateMoveBatch.AllocationInfo[0].PlacingNeedleInfo[0].Box :=LREAL_TO_UINT(Service.AllocateMoveStructure.Tobox);
	AutoAllocateJobBatch_Ctrl.AutoMode_AllocateMoveBatch.AllocationInfo[0].PlacingNeedleInfo[0].Clip:=LREAL_TO_INT(Service.AllocateMoveStructure.Clip);
	AutoAllocateJobBatch_Ctrl.AutoMode_AllocateMoveBatch.AllocationInfo[0].PlacingNeedleInfo[0].NeedleLocation :=LREAL_TO_INT(Service.AllocateMoveStructure.ToPosition);

	Service.AllocateMoveStructure.HandShake.Busy :=AutoAllocateJobBatch_Status.bBusy;
	Service.AllocateMoveStructure.HandShake.Done :=AutoAllocateJobBatch_Status.bDone;
	Service.AllocateMoveStructure.HandShake.Error :=AutoAllocateJobBatch_Status.bError;
	bAutoAllocateJobDryRun := TRUE;
END_METHOD

METHOD PRIVATE M_ManualTurnTable : BOOL
VAR_INPUT
END_VAR
_TurnTableMove.HandShake.Execute:=Service.TurnTableMove.HandShake.Execute;
_TurnTableMove.Position:=Service.TurnTableMove.Position;

Service.TurnTableMove.HandShake.Busy := _TurnTableMove.HandShake.Busy;
Service.TurnTableMove.HandShake.Done := _TurnTableMove.HandShake.Done;
Service.TurnTableMove.HandShake.Error := _TurnTableMove.HandShake.Error;
END_METHOD

METHOD PUBLIC M_ReleasePulloutAccess : BOOL
VAR_INPUT
 ControlAccess:	 E_RoundBeltControlAccess;
END_VAR
IF ControlAccess = THIS^.PulloutControlAccess THEN
		THIS^.PulloutControlAccess := E_RoundBeltControlAccess.Host;
		M_ReleasePulloutAccess := TRUE;
	ELSE
		M_ReleasePulloutAccess := FALSE;
	
END_IF
END_METHOD

METHOD PUBLIC M_ReleaseRoundBeltAccess : BOOL
VAR_INPUT
 ControlAccess:	 E_RoundBeltControlAccess;
END_VAR
IF ControlAccess = THIS^.RoundBeltControlAccess THEN
		THIS^.RoundBeltControlAccess := E_RoundBeltControlAccess.Host;
		M_ReleaseRoundBeltAccess := TRUE;
	ELSE
		M_ReleaseRoundBeltAccess := FALSE;
	
END_IF
END_METHOD

METHOD M_ResetReloadRoundBeltAction : BOOL
VAR_INPUT
END_VAR
RoundBeltMoveJob_Ctrl.Execute := FALSE;

M_ResetReloadRoundBeltAction := true; // Method end
END_METHOD

METHOD M_Resetting
IF __ISVALIDREF(Cylinder) THEN
	Clip.stCylinders.Cylinder0 REF= Cylinder.List.fbAllocateRobot_LeftClamp1;
	Clip.stCylinders.Cylinder1 REF= Cylinder.List.fbAllocateRobot_LeftClamp2;
	Clip.stCylinders.Cylinder2 REF= Cylinder.List.fbAllocateRobot_RightClamp1;
	Clip.stCylinders.Cylinder3 REF= Cylinder.List.fbAllocateRobot_RightClamp2;
	Cylinders.stCylinders.Cylinder0 REF= Cylinder.List.fbAllocateRobot_LeftVert1;
	Cylinders.stCylinders.Cylinder1 REF= Cylinder.List.fbAllocateRobot_LeftVert2;
	Cylinders.stCylinders.Cylinder2 REF= Cylinder.List.fbAllocateRobot_RightVert1;
	Cylinders.stCylinders.Cylinder3 REF= Cylinder.List.fbAllocateRobot_RightVert2;	
END_IF

M_StateComplete();
END_METHOD

METHOD PUBLIC M_StartAllocatePulloutAction : BOOL
VAR_INPUT
	CV_ForwardTime :TIME;
	CV_BackwardTIme : TIME;
	CommandType : E_PullOutConveyorCommandType; // Select PullOut conveyor command.
END_VAR
AutoPullout_Internal_Ctrl.Execute := TRUE;
AutoPullout_Internal_Info.ConveyorReverseTime := CV_BackwardTIme;
AutoPullout_Internal_Info.ConveyorRunningTime := CV_ForwardTime;
AutoPullout_Internal_Info.CommandType := CommandType;
M_StartAllocatePulloutAction := TRUE; // Method end
END_METHOD

METHOD M_StartHoming
VAR_INPUT
END_VAR
fbAllocateHome.xExecute := true;
END_METHOD

METHOD M_Starting
M_StateComplete();
END_METHOD

(* This Method is used to start round belt action : unlock pin and move to target position
	also injection the action parameter.
*)
METHOD M_StartReloadRoundBeltAtion : BOOL
VAR_INPUT
	ReloadStation : E_RoundBeltStation;
END_VAR
VAR_INST
	_ReloadStation : E_RoundBeltStation;
END_VAR
IF (ReloadStation > 12) THEN
	_ReloadStation := (ReloadStation -12 );
//	_ReloadStation := (ReloadStation -6 );
ELSE
	_ReloadStation := ReloadStation + 28;
END_IF
IF F_Even(_ReloadStation) THEN
	_ReloadStation := _ReloadStation-1;
END_IF

//IF ReloadStation > 6 THEN
//	_ReloadStation := ReloadStation -6;
//ELSE
//	_ReloadStation := ReloadStation +14;
//END_IF
//AutoRotatebelt_Internal_Ctrl.uiLatch := E_Pistons.LoadingBoxRegion;
//AutoRotatebelt_Internal_Ctrl.uiStation :=  _ReloadStation;
//AutoRotatebelt_Internal_Ctrl.Timeout := T#15S;
//AutoRotatebelt_Internal_Ctrl.bSendPressBox := FALSE; // Release allocate zone, press box cylinder in backward position
RoundBeltMoveJob_Position_FanucRobot := _ReloadStation;
RoundBeltMoveJob_Ctrl.Execute := TRUE;

M_StartReloadRoundBeltAtion := TRUE; // Method end
END_METHOD

METHOD M_StartStoragePulloutAction : BOOL
VAR_INPUT
	CV_ForwardTime :TIME;
	CV_BackwardTIme : TIME;
	CommandType : E_PullOutConveyorCommandType; // Select PullOut conveyor command.
END_VAR
RobotPullout_Internal_Ctrl.Execute := TRUE;
RobotPullout_Internal_Info.CommandType := CommandType;
RobotPullout_Internal_Info.ConveyorReverseTime := CV_BackwardTIme;
RobotPullout_Internal_Info.ConveyorRunningTime := CV_ForwardTime;
M_StartStoragePulloutAction := TRUE; // Method end
END_METHOD

METHOD M_StopAllocatePulloutAction : BOOL
VAR_INPUT
END_VAR
AutoPullout_Internal_Ctrl.Execute := FALSE;
M_StopAllocatePulloutAction := TRUE; // Methode end
END_METHOD

METHOD M_StopHoming
VAR_INPUT
END_VAR
fbAllocateHome.xExecute := False;
END_METHOD

METHOD M_Stopped
M_StateComplete();
END_METHOD

METHOD M_Stopping
M_StateComplete();
END_METHOD

METHOD M_StopStoragePulloutAction : BOOL
VAR_INPUT
END_VAR
RobotPullout_Internal_Ctrl.Execute := FALSE;
M_StopStoragePulloutAction := TRUE; //Method End
END_METHOD

METHOD M_Suspended
M_StateComplete();
END_METHOD

METHOD M_Suspending
M_StateComplete();
END_METHOD

METHOD PUBLIC M_TransCVCameraPress : BOOL
VAR_INPUT
END_VAR
VAR_INST
	
END_VAR
IF NOT TransCV_Press THEN
	//Cylinder.List.fbSameSizeCV_Press2.M_Extend();
	//Cylinder.List.fbDifferentSizeCV_Press1.M_Extend();
	TransCV_Press:=true;
END_IF
END_METHOD

METHOD PUBLIC M_TransCVCameraPress_ManualMode : BOOL
VAR_INPUT
END_VAR
IF TransCV_Press THEN
TransCV_Press := FALSE;
Cylinder.List.fbSameSizeCV_Press2.M_Retract();
Cylinder.List.fbDifferentSizeCV_Press1.M_Retract();
Cylinder.List.fbUpCV_Block1.M_Retract();
END_IF
END_METHOD

METHOD M_Undefined
M_StateComplete();
END_METHOD

METHOD M_Unholding
M_StateComplete();
END_METHOD

METHOD M_Unsuspending
M_StateComplete();
END_METHOD

END_FUNCTION_BLOCK

(* stored: Version 1.1.0.1, ProductVersion 3.1.4024.13
   POU FB_AllocateAreaWithRoundbelt: Id {4722c357-f436-40f5-9603-7e4438da9d25}, SpecialFunc None
   Folder Methods: Id {567ceadc-917a-4436-8d3c-87ac243d2566}
   Folder Private: Id {a2dbf2b1-9467-4e9e-8d1c-2ee53ae67b94}
   Folder Public: Id {0411464c-edec-4311-8959-0c7e70c946c7}
   Folder Service: Id {0f946738-f975-4678-80f0-30c3eaf451f3}
   Folder Pullout: Id {33510cf9-649a-4d09-80bf-a3852edd6021}
   Folder RoundBelt: Id {7afca88d-5485-41cf-b25c-95c8954f55a5}
   Folder States: Id {6161fa1b-6034-481c-91b9-269a6c38d9dd}
   Action A00_Service: Id {6dc1d4e2-0273-4f7f-b3c5-02c7bf6844c0}
   Action A01_RoundBeltAccessControl: Id {9a16c9c7-6b93-4040-84b9-3057330d86a4}
   Action A02_PulloutAccessControl: Id {02786782-6d97-47ca-a641-778165c2b4a0}
   Action A99_ErrorHandler: Id {a46e5a00-079e-4acb-84fa-a98399f2647e}
   Method M_Aborted: Id {f9c470e2-e837-4f99-832c-94f4bf162e68}
   Method M_Aborting: Id {f47ed5d0-d581-4899-a335-17f7b5663966}
   Method M_ActiveRoundBeltInternalCtrl: Id {6383c384-733f-448a-af39-61c53bd0511a}
   Method M_AutoAllocatingBatch: Id {78ee68fe-a3ae-473c-9c05-2e1ae9f2e998}
   Method M_AutoAllocatingBatch_Reverse: Id {32353bb2-171c-4822-be0e-c5035ae517d7}
   Method M_AutoAllocatingBatch_Simple: Id {cbb871bb-237a-4e42-9688-397726b21265}
   Method M_AutoTurnTable: Id {f75f7c7d-482b-41a5-a75f-40f52d49dc4c}
   Method M_CheckAxesHomed: Id {b35024de-bb1c-4394-9395-73defc78c724}
   Method M_Clearing: Id {562fd765-7485-4a82-ad8c-2302e5773406}
   Method M_Complete: Id {b794b69c-9b74-45a7-b7e9-90266dcd9ba9}
   Method M_Completing: Id {38eb0607-073b-48a9-aa3b-ecccbe48f662}
   Method M_Execute: Id {baa71317-3ff7-4b6b-969f-b75b5d9f57f5}
   Method M_GetPulloutAccess: Id {ccaa9946-2575-44d9-8e45-317018f1962b}
   Method M_GetRoundBeltAccess: Id {90ae85e4-3deb-4b75-b56f-224a2ad296d9}
   Method M_Held: Id {22d96dbd-4aab-4e54-b6ce-fc857f6ce98c}
   Method M_Holding: Id {f27d6b7b-05c5-45f7-a0fb-68acce83e3d8}
   Method M_Idle: Id {5d6418ec-5854-4049-82a5-89dffe187b4b}
   Method M_InactiveRoundBeltInternalCtrl: Id {134ac148-980a-4a36-8d6a-23d797a19726}
   Method M_ManualAllocating: Id {389ed1a5-e4d2-47be-9c6b-2144473f1d9f}
   Method M_ManualTurnTable: Id {65b94d0c-2090-47fe-b70a-f2f4b0f4a272}
   Method M_ReleasePulloutAccess: Id {4f5bc646-5dbd-4ce4-a828-74a5f6d4cdbf}
   Method M_ReleaseRoundBeltAccess: Id {ab6b25d9-94ba-4c5f-bbc8-f977ff5d7afc}
   Method M_ResetReloadRoundBeltAction: Id {9a5f7dec-a67e-4f7b-8a2b-0419ec8fb38f}
   Method M_Resetting: Id {7510f6ff-5c2a-4f62-8abe-ee2e640016d2}
   Method M_StartAllocatePulloutAction: Id {37aa1ecf-5cf1-4e3d-acb8-8e3d2ba00b09}
   Method M_StartHoming: Id {620fd941-f4b2-4243-a20a-47ba680e35d9}
   Method M_Starting: Id {3a8261d0-5827-46bd-9f71-a59c36e02c06}
   Method M_StartReloadRoundBeltAtion: Id {2e4beba3-6217-472d-a192-467f8534f6ad}
   Method M_StartStoragePulloutAction: Id {8dc4f638-5d0d-4a69-b402-ecd0f2373a12}
   Method M_StopAllocatePulloutAction: Id {2c14123f-718b-4b06-80ab-923ef7993357}
   Method M_StopHoming: Id {d8160e10-8ca9-4893-a438-0b0b93d2874b}
   Method M_Stopped: Id {39e500ba-92f0-41c1-80a1-e71edaa73f13}
   Method M_Stopping: Id {5caef25a-f20a-4282-b342-71351aa35822}
   Method M_StopStoragePulloutAction: Id {a3597a0f-e44f-4bdd-91d5-1302fcc65662}
   Method M_Suspended: Id {f96c1e03-e8e6-4bb0-a56b-b26b4d2a2631}
   Method M_Suspending: Id {f48f74b9-0baa-49d4-9206-553db8a3e572}
   Method M_TransCVCameraPress: Id {5f84a7db-a711-4a0d-8fba-6048be8fe807}
   Method M_TransCVCameraPress_ManualMode: Id {681d7f6b-44b9-4e2d-9945-14a2837af570}
   Method M_Undefined: Id {4ce511e2-d0e3-4d03-afd6-a4a676bdd5eb}
   Method M_Unholding: Id {b755af47-9939-4109-bae2-60553ccf9e78}
   Method M_Unsuspending: Id {5b13d8ab-89a0-4a49-9578-02effb5e958f} *)
